TYPE E_TransportControlRemoveTU_Emulation :
(**************************************************************************************
 * 	Application		:	BoxControl Framework
 *	Revision		:	$Revision: 404529 $
 *	Revision date	:	$Date: 2018-04-23 08:21:38 +0200 (Mo., 23 Apr 2018) $
 *	Last changed by	:	$Author: b7bolm $
 *	URL				:	$URL: http://almscdc.swisslog.com/repo/SWPD/Development/BoxControlFramework/20_Release/trunk/01_Software/BCF/BCF/JumpStart/20_Product/11_Emu/12_E_Functions/10_Lib/10_Conv/10_Functions/01_DUTs/E_TransportControlRemoveTU_Emulation.TcDUT $
 *
 *	Purpose			:	TransportControl remove TU type definition
 *
 * ------------------------------------------------------------------------------------
 *	Copyright Swisslog [IP AG], Switzerland. All rights reserved.
 * 
 * ------------------------------------------------------------------------------------
 *	
 * 	Revision History: 
 *
 * 	VERSION			DATE			INITIALS			DESCRIPTION
 *	0.1				01.01.2001		swl					Example
 *
 **************************************************************************************)	
(
	IDLE_REMOVE_TU, // Location ready to remove a TU 
	START_REMOVE_TU, // Start removing a TU 
	BUSY_REMOVE_TU // Removing TU's 
);
END_TYPE

(* stored: Version 1.1.0.1, ProductVersion 3.1.4022.12
   DUT E_TransportControlRemoveTU_Emulation: Id {e2f3143b-daee-44c0-98f9-a053ebad557a} *)
